// TIA Portal V16 export
// export: Created 2024-09-05T17:39:24.7159148Z, ExportSetting WithDefaults, DisplayName Totally Integrated Automation Portal, DisplayVersion V16 Update 6, DisplayName TIA Portal Version Control Interface, DisplayVersion V16 Update 2, DisplayName TIA Portal Openness, DisplayVersion V16 Update 6, DisplayName STEP 7 Professional, DisplayVersion V16 Update 6, DisplayName STEP 7 Safety, DisplayVersion V16, DisplayName WinCC Advanced, DisplayVersion V16 Update 6
DATA_BLOCK "1. DMC_setConnection_DB"   // DB2002
AUTHOR : bartz
VERSION : 0.1
// stored: AutoNumber false, DBAccessibleFromOPCUA true, InstanceOfName 1. DMC_setConnection, InstanceOfType FB
"1. DMC_setConnection"
   // VAR
   //    Connection : Struct
   //       IPAddress : WString;
   //       ServerPort : WString;
   //       PlantID : WString;
   //       PLC_ID : WString;
   //       OperationMode : Bool;
   //    END_STRUCT;
   //    Controllers : Struct
   //       opcUaConnect : Bool;
   //       opcUaMethodCall : Bool;
   //       opcUaMethodIndex : SInt;
   //       opcUaConnected { S7_SetPoint := 'True'} : Bool;
   //       opcUaDone : Bool;
   //       opcUaBusy : Bool;
   //       opcUaError : Bool;
   //       opcUaStatus : Word;
   //       opcUaDiagnostics : "typeFbDiagnostics";
   //    END_STRUCT;
   //    Auxiliar : Struct
   //       endpointTemp : String[254];
   //       idx : Int;
   //       timeout : Bool;
   //       life : Bool;
   //       closedRequested : Bool;
   //       tryAgain : Bool;
   //       attempts : Int;
   //    END_STRUCT;
   //    Timers : Struct
   //       timeoutCallMethod : TON_TIME;
   //       forceReconnection { S7_SetPoint := 'True'} : TON_TIME;
   //       tryAgain { S7_SetPoint := 'True'} : TON_TIME;
   //    END_STRUCT;
   //    CallBuffer : Array[0..9] of Bool;
   // END_VAR
BEGIN
END_DATA_BLOCK
